(* IEC 61131-3 sources: volt/packages/volt-lsp-iec/test-corpus/pro2193/Device/Plc Logic/Application/09 Misc/Library Manager/L_EtcSlaveConfig_i750, 13 files *)

(* ---- PARASAVE_STATE_I900.dut ---- *)
TYPE PARASAVE_STATE_I900 :
(
	SAVE_INITIALIZE,
	SAVE_WAIT_GET_SLAVE_STATE,
	SAVE_SAVING,
	SAVE_ERROR,
	SAVE_DONE
);
END_TYPE

(* ---- RESTART_FIRMWARE_STATE_I750.dut ---- *)
TYPE RESTART_FIRMWARE_STATE_I750 :
(
	RSFWI700_INITIALIZE,
	RSFWI700_WAIT_FOR_GETSTATE_FINISHED,
	RSFWI700_WAIT_FOR_RESTART2_DONE,
	RSFWI700_ERROR,
	RSFWI700_DONE
);
END_TYPE

(* ---- GETBOOLEANPROPERTY.pou ---- *)
FUNCTION GETBOOLEANPROPERTY : BOOL
VAR_INPUT
	STKEY : WSTRING;
END_VAR
END_FUNCTION

(* ---- GETCOMPANY.pou ---- *)
FUNCTION GETCOMPANY : WSTRING
END_FUNCTION

(* ---- GETNUMBERPROPERTY.pou ---- *)
FUNCTION GETNUMBERPROPERTY : DINT
VAR_INPUT
	STKEY : WSTRING;
END_VAR
END_FUNCTION

(* ---- GETTEXTPROPERTY.pou ---- *)
FUNCTION GETTEXTPROPERTY : WSTRING
VAR_INPUT
	STKEY : WSTRING;
END_VAR
END_FUNCTION

(* ---- GETTEXTPROPERTY2.pou ---- *)
FUNCTION GETTEXTPROPERTY2 : POINTER TO WSTRING
VAR_INPUT
	STKEY : WSTRING;
END_VAR
END_FUNCTION

(* ---- GETTITLE.pou ---- *)
FUNCTION GETTITLE : WSTRING
END_FUNCTION

(* ---- GETVERSION.pou ---- *)
FUNCTION GETVERSION : VERSION
END_FUNCTION

(* ---- GETVERSIONPROPERTY.pou ---- *)
FUNCTION GETVERSIONPROPERTY : VERSION
VAR_INPUT
	STKEY : WSTRING;
END_VAR
END_FUNCTION

(* ---- ETCFIRMWAREDOWNLOAD_I750.pou ---- *)
FUNCTION_BLOCK ETCFIRMWAREDOWNLOAD_I750 EXTENDS EtcFirmwareDownload_i700
VAR
	READCURRENTAXIS : L_ETC_CoE_SdoRead;
	BYAXISTYPE : BYTE;
	RESTARTSTATEI750 : RESTART_FIRMWARE_STATE_I750 := RSFW_INITIALIZE;
	ISAXISB : BOOL;
END_VAR
END_FUNCTION_BLOCK

METHOD CALLBEFOREGETVERSION
END_METHOD

METHOD GETFILENAMEFORFOETRANSFER : CAA_FILENAME
END_METHOD

METHOD GETTIMEOUTFORFOEFIRMWARETRANSFER : UDINT
END_METHOD

METHOD ISFIRMWAREDOWNLOADTYPEI750 : BOOL
END_METHOD

METHOD MUSTCALLBEFOREGETVERSION : BOOL
END_METHOD

METHOD RESETALLSIGNALS : BOOL
END_METHOD

METHOD RESTARTTYPE_I750
END_METHOD

METHOD SHOULDUPDATE : CHECKVERSION_FIRMWARE_RESULT
VAR_INPUT
	STARGETVERSIONMAJOR : STRING(10);
	STARGETVERSIONMINOR : STRING(10);
	STARGETVERSIONPATCHLEVEL : STRING(10);
	STARGETVERSIONBUILDNUMBER : STRING(10);
	SSLAVEVERSIONMAJOR : STRING(10);
	SSLAVEVERSIONMINOR : STRING(10);
	SSLAVEVERSIONPATCHLEVEL : STRING(10);
	SSLAVEVERSIONBUILDNUMBER : STRING(10);
	BYFWDLMODE : BYTE;
END_VAR
END_METHOD

(* ---- ETCSAVEPARAMETERSET_I750.pou ---- *)
FUNCTION_BLOCK ETCSAVEPARAMETERSET_I750 EXTENDS L_SUDP_UpDownload
VAR
	PETCDEV : POINTER TO ETCSlave;
	ECONTROL : L_SUDP_Control;
	A : INT;
	BYOLDVALUEOFCONTROLINPUT : L_SUDP_Control;
	SAVESTATE : PARASAVE_STATE_I900 := PARASAVE_STATE_I900.SAVE_INITIALIZE;
	GETSLAVESTATE : L_ETC_GetSlaveState;
	GETETCMASTERDIAGNOSTIC : L_ETC_GetMasterDiagnostic;
	SDOWR : L_ETC_CoE_SdoWrite;
	PARSAVEVALUE : BYTE := 1;
	ESAVEERROR : L_SUDP_ErrorCodes;
END_VAR
END_FUNCTION_BLOCK

METHOD INITIALIZE
VAR_INPUT
	PETCREMDEV : POINTER TO L_ETCSlave;
END_VAR
END_METHOD

METHOD SAVE
END_METHOD

(* ---- L_ETCSLAVE_I750.pou ---- *)
FUNCTION_BLOCK L_ETCSLAVE_I750
VAR_OUTPUT
	PETCSLAVE : POINTER TO ETCSlave;
END_VAR
VAR
	ETCSLAVE : ETCSlave;
	M_HLEMACCESS_I750 : RTS_IEC_HANDLE;
	PARSETXFER : L_ECC_i700.EtcConfigParaXfer_i700;
	FIRMWAREDOWNLOAD : EtcFirmwareDownload_i750;
	PARSETUPLOAD : L_ECC_i700.EtcConfigParaUpload_i700;
	ISMANDATORY : BOOL;
	ISPRESENT : BOOL;
	MODULEHANDLER : L_IMHP_IModuleHandler;
END_VAR
END_FUNCTION_BLOCK

METHOD CYCLICCALL : UDINT
END_METHOD

METHOD FB_EXIT : BOOL
VAR_INPUT
	BINCOPYCODE : BOOL;
END_VAR
END_METHOD

METHOD FB_INIT : BOOL
VAR_INPUT
	BINITRETAINS : BOOL;
	BINCOPYCODE : BOOL;
END_VAR
END_METHOD

METHOD INITIALIZE : UDINT
VAR_INPUT
	WMODULETYPE : UINT;
	DWINSTANCE : UDINT;
	PCONNECTOR : POINTER TO IoConfigConnector;
END_VAR
END_METHOD
